FUNCTION_BLOCK GET_CHAN_INFO (* Loads channel with the specified symbolic name *)
  (* Standard: 61499-2 *)
  (* Version 0.0, 2011-09-22, 4DIAC-IDE, 4DIAC-Consortium *)
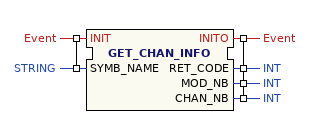
  EVENT_INPUT
    INIT WITH SYMB_NAME;
  END_EVENT
  EVENT_OUTPUT
    INITO WITH RET_CODE, MOD_NB, CHAN_NB; (* Initialization Confirm *)
  END_EVENT
  VAR_INPUT
    SYMB_NAME : STRING; (* Symbolic channel name *)
  END_VAR
  VAR_OUTPUT
    RET_CODE : INT; (* Return Code *)
    MOD_NB : INT; (* Module number *)
    CHAN_NB : INT; (* Channel number *)
  END_VAR
  SERVICE APPLICATION/RESOURCE (* Loads channel with the specified symbolic name *)
    SEQUENCE normal_establishment
      APPLICATION.INIT+(PARAMS) -> APPLICATION.INITO+(PARAMS);
    END_SEQUENCE
    SEQUENCE unsuccessful_establishment
      APPLICATION.INIT+(PARAMS) -> APPLICATION.INITO-(STATUS);
    END_SEQUENCE
    SEQUENCE request_confirm
      APPLICATION.REQ+(SD) -> APPLICATION.CNF+(RD);
    END_SEQUENCE
    SEQUENCE request_inhibited
      APPLICATION.REQ-(SD) -> APPLICATION.CNF-(STATUS);
    END_SEQUENCE
    SEQUENCE request_error
      APPLICATION.REQ+(SD) -> APPLICATION.CNF-(STATUS);
    END_SEQUENCE
    SEQUENCE indication_inhibited
      RESOURCE.indicate(RD,QI=FALSE) -> RESOURCE.inhibited();
    END_SEQUENCE
    SEQUENCE application_initiated_termination
      APPLICATION.INIT-() -> APPLICATION.INITO-(STATUS);
    END_SEQUENCE
    SEQUENCE resource_initiated_termination
      -> APPLICATION.INITO-(STATUS);
    END_SEQUENCE
  END_SERVICE
END_FUNCTION_BLOCK
